// TIA Portal V18 export
FUNCTION "AHURegsAndTargetStatesInPreComfortOpMode" : Void   // FC60032, LAD
{ S7_Optimized_Access := 'TRUE' }
VERSION : 0.1
// Operation Modes                                                 Unit State
// 0                                                                             0=Stopped
// 1                                                                             1=Checking-up  
// 2 PreComfort                                                        2=Preheating
//                                                                                 3=Starting 
//                                                                                 4=RecirculatingOperation (Protection)
//                                                                                 5=Sustained Mode (Economy)
//                                                                                 6=Sustained Mode (PreComfort setpoints) 
//                                                                                 Not 7=Comfort  operation
//                                                                                 Not 8=Night Cooling
//                                                                                 9=Stopping
//                                                                                 10=Blocking
//                                                                                 11=FrostProtecting
// stored: AutoNumber false, IsIECCheckEnabled false, SetENOAutomatically false, UDAEnableTagReadback false
   VAR_INPUT
      iUnitID : Int;
      cActualOpMode : Byte;
      cHeatingRegCfg : Byte;
      cCoolingRegCfg : Byte;
      cIAQRegCfg : Byte;
      cBuildingdPRegCfg : Byte;
   END_VAR
   VAR_OUTPUT
      cTargetState : Byte;
      cHeatingRegState : Byte;
      cCoolingRegState : Byte;
      cIAQRegState : Byte;
      cBuildingdPRegState : Byte;
   END_VAR
   VAR_TEMP
      SHTargetState : Byte;
      SCTargetState : Byte;
      SIAQTargetState : Byte;
      SdPTargetState : Byte;
   END_VAR
BEGIN

REGION Network 1: Sustained Heating
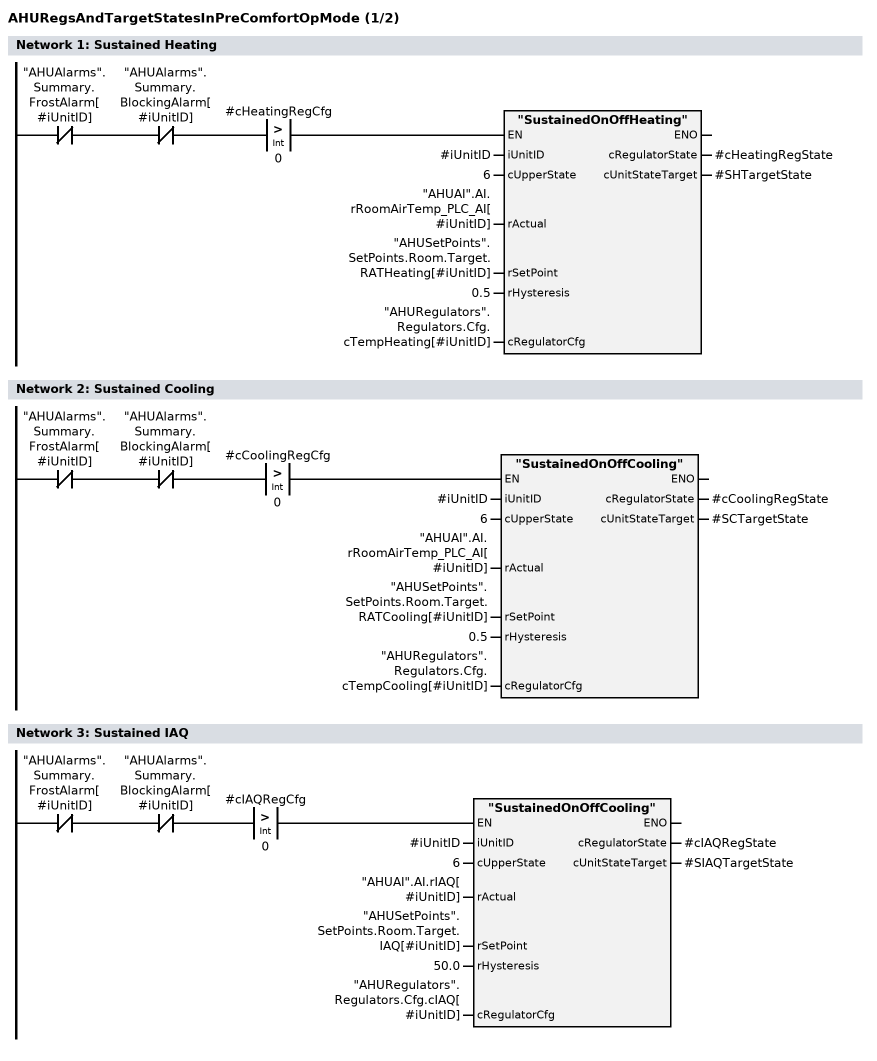
   RUNG wire#powerrail
      I_Contact( "AHUAlarms".Summary.FrostAlarm[#iUnitID] )
      I_Contact( "AHUAlarms".Summary.BlockingAlarm[#iUnitID] )
      { S7_Templates := "SrcType := Int" } GT_Contact(in1 := #cHeatingRegCfg, in2 := 0)
      "SustainedOnOffHeating"(iUnitID := #iUnitID, cUpperState := 6, rActual := "AHUAI".AI.rRoomAirTemp_PLC_AI[#iUnitID], rSetPoint := "AHUSetPoints".SetPoints.Room.Target.RATHeating[#iUnitID], rHysteresis := 0.5, cRegulatorCfg := "AHURegulators".Regulators.Cfg.cTempHeating[#iUnitID], cRegulatorState => #cHeatingRegState, cUnitStateTarget => #SHTargetState)
   END_RUNG
   // the same network as SCL:
   IF NOT "AHUAlarms".Summary.FrostAlarm[#iUnitID] AND NOT "AHUAlarms".Summary.BlockingAlarm[#iUnitID] AND (#cHeatingRegCfg > 0) THEN
       "SustainedOnOffHeating"(iUnitID := #iUnitID,
                               cUpperState := 6,
                               rActual := "AHUAI".AI.rRoomAirTemp_PLC_AI[#iUnitID],
                               rSetPoint := "AHUSetPoints".SetPoints.Room.Target.RATHeating[#iUnitID],
                               rHysteresis := 0.5,
                               cRegulatorCfg := "AHURegulators".Regulators.Cfg.cTempHeating[#iUnitID],
                               cRegulatorState => #cHeatingRegState,
                               cUnitStateTarget => #SHTargetState);
   END_IF;
END_REGION

REGION Network 2: Sustained Cooling
   RUNG wire#powerrail
      I_Contact( "AHUAlarms".Summary.FrostAlarm[#iUnitID] )
      I_Contact( "AHUAlarms".Summary.BlockingAlarm[#iUnitID] )
      { S7_Templates := "SrcType := Int" } GT_Contact(in1 := #cCoolingRegCfg, in2 := 0)
      "SustainedOnOffCooling"(iUnitID := #iUnitID, cUpperState := 6, rActual := "AHUAI".AI.rRoomAirTemp_PLC_AI[#iUnitID], rSetPoint := "AHUSetPoints".SetPoints.Room.Target.RATCooling[#iUnitID], rHysteresis := 0.5, cRegulatorCfg := "AHURegulators".Regulators.Cfg.cTempCooling[#iUnitID], cRegulatorState => #cCoolingRegState, cUnitStateTarget => #SCTargetState)
   END_RUNG
   // the same network as SCL:
   IF NOT "AHUAlarms".Summary.FrostAlarm[#iUnitID] AND NOT "AHUAlarms".Summary.BlockingAlarm[#iUnitID] AND (#cCoolingRegCfg > 0) THEN
       "SustainedOnOffCooling"(iUnitID := #iUnitID,
                               cUpperState := 6,
                               rActual := "AHUAI".AI.rRoomAirTemp_PLC_AI[#iUnitID],
                               rSetPoint := "AHUSetPoints".SetPoints.Room.Target.RATCooling[#iUnitID],
                               rHysteresis := 0.5,
                               cRegulatorCfg := "AHURegulators".Regulators.Cfg.cTempCooling[#iUnitID],
                               cRegulatorState => #cCoolingRegState,
                               cUnitStateTarget => #SCTargetState);
   END_IF;
END_REGION

REGION Network 3: Sustained IAQ
   RUNG wire#powerrail
      I_Contact( "AHUAlarms".Summary.FrostAlarm[#iUnitID] )
      I_Contact( "AHUAlarms".Summary.BlockingAlarm[#iUnitID] )
      { S7_Templates := "SrcType := Int" } GT_Contact(in1 := #cIAQRegCfg, in2 := 0)
      "SustainedOnOffCooling"(iUnitID := #iUnitID, cUpperState := 6, rActual := "AHUAI".AI.rIAQ[#iUnitID], rSetPoint := "AHUSetPoints".SetPoints.Room.Target.IAQ[#iUnitID], rHysteresis := 50.0, cRegulatorCfg := "AHURegulators".Regulators.Cfg.cIAQ[#iUnitID], cRegulatorState => #cIAQRegState, cUnitStateTarget => #SIAQTargetState)
   END_RUNG
   // the same network as SCL:
   IF NOT "AHUAlarms".Summary.FrostAlarm[#iUnitID] AND NOT "AHUAlarms".Summary.BlockingAlarm[#iUnitID] AND (#cIAQRegCfg > 0) THEN
       "SustainedOnOffCooling"(iUnitID := #iUnitID,
                               cUpperState := 6,
                               rActual := "AHUAI".AI.rIAQ[#iUnitID],
                               rSetPoint := "AHUSetPoints".SetPoints.Room.Target.IAQ[#iUnitID],
                               rHysteresis := 50.0,
                               cRegulatorCfg := "AHURegulators".Regulators.Cfg.cIAQ[#iUnitID],
                               cRegulatorState => #cIAQRegState,
                               cUnitStateTarget => #SIAQTargetState);
   END_IF;
END_REGION

REGION Network 4: Sustained BuildingdP
   // !!!!Додати опрацьовку Сили вітриу з погодної станції
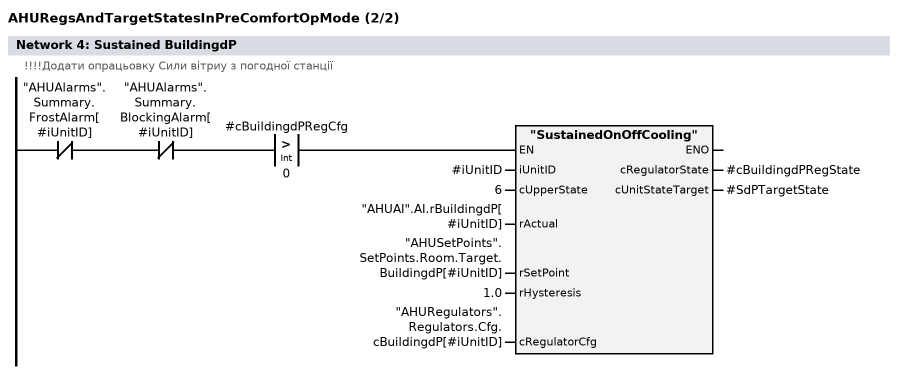
   RUNG wire#powerrail
      I_Contact( "AHUAlarms".Summary.FrostAlarm[#iUnitID] )
      I_Contact( "AHUAlarms".Summary.BlockingAlarm[#iUnitID] )
      { S7_Templates := "SrcType := Int" } GT_Contact(in1 := #cBuildingdPRegCfg, in2 := 0)
      "SustainedOnOffCooling"(iUnitID := #iUnitID, cUpperState := 6, rActual := "AHUAI".AI.rBuildingdP[#iUnitID], rSetPoint := "AHUSetPoints".SetPoints.Room.Target.BuildingdP[#iUnitID], rHysteresis := 1.0, cRegulatorCfg := "AHURegulators".Regulators.Cfg.cBuildingdP[#iUnitID], cRegulatorState => #cBuildingdPRegState, cUnitStateTarget => #SdPTargetState)
   END_RUNG
   // the same network as SCL:
   IF NOT "AHUAlarms".Summary.FrostAlarm[#iUnitID] AND NOT "AHUAlarms".Summary.BlockingAlarm[#iUnitID] AND (#cBuildingdPRegCfg > 0) THEN
       "SustainedOnOffCooling"(iUnitID := #iUnitID,
                               cUpperState := 6,
                               rActual := "AHUAI".AI.rBuildingdP[#iUnitID],
                               rSetPoint := "AHUSetPoints".SetPoints.Room.Target.BuildingdP[#iUnitID],
                               rHysteresis := 1.0,
                               cRegulatorCfg := "AHURegulators".Regulators.Cfg.cBuildingdP[#iUnitID],
                               cRegulatorState => #cBuildingdPRegState,
                               cUnitStateTarget => #SdPTargetState);
   END_IF;
END_REGION

REGION Network 5 (SCL)
   #SHTargetState := MAX(IN1 := #SHTargetState, IN2 := #SCTargetState);
   #SIAQTargetState := MAX(IN1 := #SIAQTargetState, IN2 := #SdPTargetState);
   #cTargetState := MAX(IN1 := #SIAQTargetState, IN2 := #SHTargetState);
END_REGION
END_FUNCTION
